TYPE Celsius EXTENDS TerminalStatus :
STRUCT
    _ : REAL;
END_STRUCT
END_TYPE

(* stored: Version 1.1.0.1, ProductVersion 3.1.4024.4
   DUT Celsius: Id {ab40127f-c650-4882-b09d-61cba668f119} *)
